// TwinCAT 3 PLC project AssertionTests
// ProgramVersion: 3.1.4023.0
// libraries:
//   CNM_AbstractObject, * (ekvip automation GmbH)
//   CNM_AssertionInterfaceLib, * (ekvip automation GmbH)
//   CNM_AssertionInterfaceTests, * (ekvip automation GmbH)
//   CNM_ReturnTypes, * (ekvip automation GmbH)
//   Tc2_CncBase, * (Beckhoff Automation GmbH)
//   Tc2_CncHli, * (Beckhoff Automation GmbH)
//   Tc2_Standard, * (Beckhoff Automation GmbH)
//   Tc2_System, * (Beckhoff Automation GmbH)
//   Tc3_Module, * (Beckhoff Automation GmbH)
//   TcUnit, * (www.tcunit.org)
// project tree:
//   ConcreteAssertions/ ConcreteAssertions.TcPOU
//   MainTask/ MAIN.TcPOU, PlcTask.TcTTO
// real-time tasks:
//   TASK PlcTask: cycle T#10ms, priority 20, ADS port 350

CONFIGURATION AssertionTests
    RESOURCE PLC ON TwinCAT3
        TASK PlcTask(INTERVAL := T#10ms, PRIORITY := 20);
        PROGRAM MAIN WITH PlcTask : MAIN;
    END_RESOURCE
END_CONFIGURATION

// ---- MainTask/MAIN.TcPOU
PROGRAM MAIN
VAR
	concrete				:ConcreteAssertions();
	tests					:CNM_AssertionInterfaceTests.AssertionTester(concrete);
END_VAR

TcUnit.RUN_IN_SEQUENCE();

END_PROGRAM

// ---- ConcreteAssertions/ConcreteAssertions.TcPOU
FUNCTION_BLOCK ConcreteAssertions EXTENDS CNM_AssertionInterfaceLib.AbstractAssertor IMPLEMENTS CNM_AssertionInterfaceTests.IAssertorContainer
VAR
	wrongAssertion	:BOOL;
END_VAR

METHOD assertionWasWrong
VAR_INPUT
	caller			:CNM_AbstractObject.IObject;
	message			:AssertMessage;
	additionalText	:Tc2_System.T_MaxString;
END_VAR
THIS^.wrongAssertion := TRUE;
END_METHOD

PROPERTY assertor : CNM_AssertionInterfaceTests.CNM_AssertionInterfaceLib.IAssertor
GET
assertor := THIS^;
END_GET
END_PROPERTY

PROPERTY className : CNM_AbstractObject.ClassName
GET
className := 'ConcreteAssertions';
END_GET
END_PROPERTY

METHOD resetAssertor
THIS^.wasAssertionWrong := FALSE;
END_METHOD

PROPERTY wasAssertionWrong : BOOL
GET
wasAssertionWrong := THIS^.wrongAssertion;
END_GET
SET
THIS^.wrongAssertion := wasAssertionWrong;
END_SET
END_PROPERTY

END_FUNCTION_BLOCK
